// TIA Portal V17 export
// export: Created 2025-03-05T08:03:14.3285164Z, ExportSetting WithDefaults, DisplayName Totally Integrated Automation Portal, DisplayVersion V17 Update 8, DisplayName TIA Portal Openness, DisplayVersion V17 Update 8, DisplayName TIA Portal Version Control Interface, DisplayVersion V17, DisplayName SINAMICS Startdrive Advanced, DisplayVersion V17 SP2, DisplayName SINAMICS Startdrive G110M, G120, G120C, G120D, G120P, G115D, DisplayVersion V17 SP2, DisplayName SINAMICS Startdrive G130, G150, S120, S150, SINAMICS MV, S210, DisplayVersion V17 SP2, DisplayName STEP 7 Professional, DisplayVersion V17 Update 8, DisplayName SINUMERIK ONE STEP 7 Toolbox, DisplayVersion V17 Update 12, DisplayName SINUMERIK 840D sl STEP 7 Toolbox, DisplayVersion V17 Update 12, DisplayName STEP 7 Safety, DisplayVersion V17 Update 6, DisplayName WinCC Advanced, DisplayVersion V17 Update 8
FUNCTION_BLOCK "FB22102_POWDER_FLOW_SENSOR"   // FB22102, LAD
TITLE = FB22102 POWDER FLOW SENSOR
{ S7_Optimized_Access := 'FALSE' }
VERSION : 0.1
// stored: AutoNumber false, IsIECCheckEnabled false, SetENOAutomatically false, UDAEnableTagReadback false
   VAR_INPUT
      iANALOG_INPUT : UInt;
   END_VAR
   VAR_OUTPUT
      oPOWDER_FLOW_ON : Bool;
      oWARNING_LIMIT : Bool;
   END_VAR
   VAR DB_SPECIFIC
      OUTPUT : Struct
         VALUE : Real;
      END_STRUCT;
      INPUT_SETTINGS : Struct
         LOW_RANGE : Real;
         HIGH_RANGE : Real;
         LOW_LIM_TO_FLOW_ON : Real;
         UNIT_NUMBER : Int;
         HOPPER_NUMBER : Int;
      END_STRUCT;
      ALARM_SETTINGS : Struct
         WARN_LIMIT_LOW : Real;
         WARN_LIMIT_HIGH : Real;
         ERROR_CONFIGURATION : Bool;
      END_STRUCT;
      LOG : Struct
         SPARE : Bool;
      END_STRUCT;
   END_VAR
   VAR_TEMP
      DB_NUMBER : DInt;
      NORM_VALUE : Real;
   END_VAR
BEGIN

NETWORK
TITLE = READ INSTANCE DB NUMBER
      L     DINO;
      +     10#800000;
      T     #DB_NUMBER;

REGION Network 2: NORM AND SCALE ANALOG INPUT
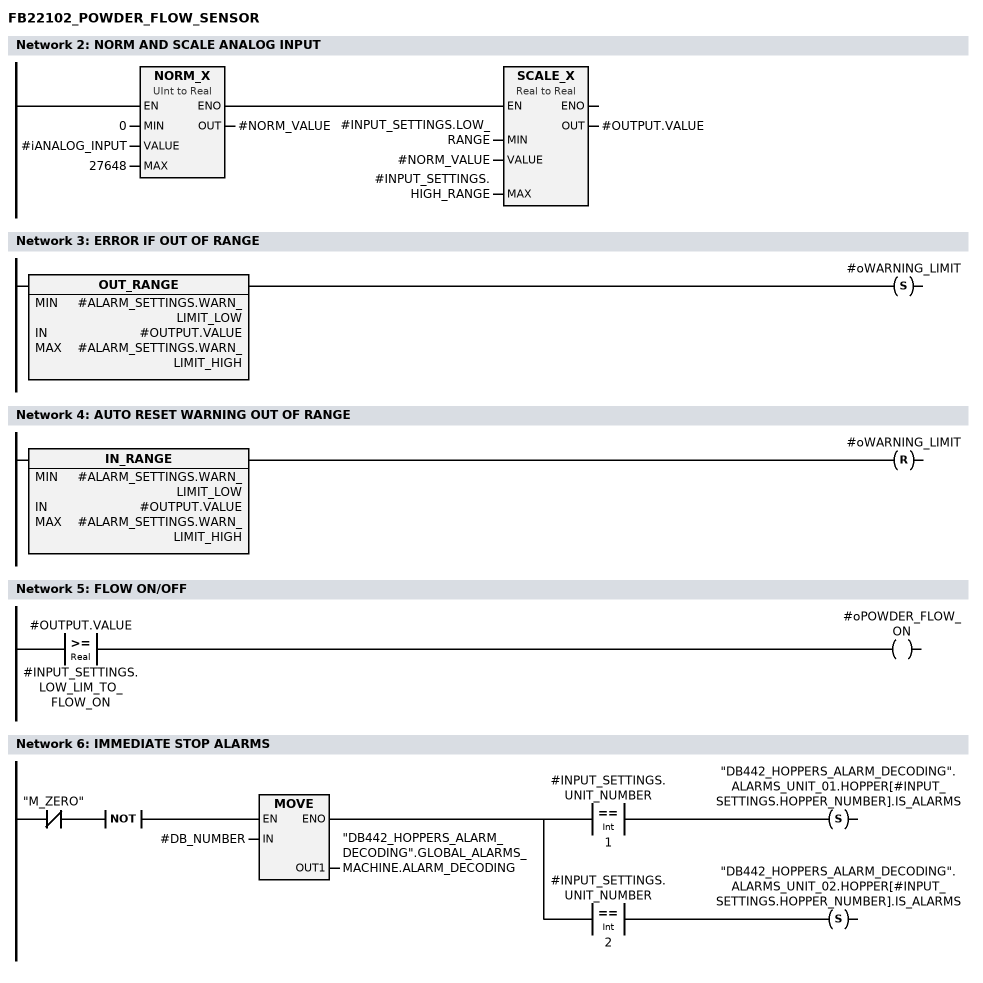
   RUNG wire#powerrail
      { S7_Templates := "[SrcType := UInt, DestType := Real]" } Normalize(min := 0, value := #iANALOG_INPUT, max := 27648, out => #NORM_VALUE)
      { S7_Templates := "[SrcType := Real, DestType := Real]" } Scale(min := #INPUT_SETTINGS.LOW_RANGE, value := #NORM_VALUE, max := #INPUT_SETTINGS.HIGH_RANGE, out => #OUTPUT.VALUE)
   END_RUNG
   // the same network as SCL:
   #NORM_VALUE := NORM_X(MIN := 0, VALUE := #iANALOG_INPUT, MAX := 27648);
   #OUTPUT.VALUE := SCALE_X(MIN := #INPUT_SETTINGS.LOW_RANGE, VALUE := #NORM_VALUE, MAX := #INPUT_SETTINGS.HIGH_RANGE);
END_REGION

REGION Network 3: ERROR IF OUT OF RANGE
   IF (#OUTPUT.VALUE < #ALARM_SETTINGS.WARN_LIMIT_LOW) OR (#OUTPUT.VALUE > #ALARM_SETTINGS.WARN_LIMIT_HIGH) THEN
       #oWARNING_LIMIT := TRUE;
   END_IF;
END_REGION

REGION Network 4: AUTO RESET WARNING OUT OF RANGE
   RUNG wire#powerrail
      { S7_Templates := "SrcType := Real" } InRange(min := #ALARM_SETTINGS.WARN_LIMIT_LOW, in := #OUTPUT.VALUE, max := #ALARM_SETTINGS.WARN_LIMIT_HIGH)
      R_Coil( #oWARNING_LIMIT )
   END_RUNG
   // the same network as SCL:
   IF (#ALARM_SETTINGS.WARN_LIMIT_LOW <= #OUTPUT.VALUE) AND (#OUTPUT.VALUE <= #ALARM_SETTINGS.WARN_LIMIT_HIGH) THEN
       #oWARNING_LIMIT := FALSE;
   END_IF;
END_REGION

REGION Network 5: FLOW ON/OFF
   RUNG wire#powerrail
      { S7_Templates := "SrcType := Real" } GE_Contact(in1 := #OUTPUT.VALUE, in2 := #INPUT_SETTINGS.LOW_LIM_TO_FLOW_ON)
      Coil( #oPOWDER_FLOW_ON )
   END_RUNG
   // the same network as SCL:
   #oPOWDER_FLOW_ON := #OUTPUT.VALUE >= #INPUT_SETTINGS.LOW_LIM_TO_FLOW_ON;
END_REGION

REGION Network 6: IMMEDIATE STOP ALARMS
   RUNG wire#powerrail
      I_Contact( "M_ZERO" )
      Not()
      { S7_GenerateENO := "TRUE" } Move(in := #DB_NUMBER, out1 => "DB442_HOPPERS_ALARM_DECODING".GLOBAL_ALARMS_MACHINE.ALARM_DECODING)
      wire#w1
      { S7_Templates := "SrcType := Int" } EQ_Contact(in1 := #INPUT_SETTINGS.UNIT_NUMBER, in2 := 1)
      S_Coil( "DB442_HOPPERS_ALARM_DECODING".ALARMS_UNIT_01.HOPPER[#INPUT_SETTINGS.HOPPER_NUMBER].IS_ALARMS )
   END_RUNG
   RUNG wire#w1
      { S7_Templates := "SrcType := Int" } EQ_Contact(in1 := #INPUT_SETTINGS.UNIT_NUMBER, in2 := 2)
      S_Coil( "DB442_HOPPERS_ALARM_DECODING".ALARMS_UNIT_02.HOPPER[#INPUT_SETTINGS.HOPPER_NUMBER].IS_ALARMS )
   END_RUNG
   // the same network as SCL:
   // ENO of a box is taken as its EN; it also drops when the box reports an error
   IF NOT (NOT "M_ZERO") THEN
       "DB442_HOPPERS_ALARM_DECODING".GLOBAL_ALARMS_MACHINE.ALARM_DECODING := #DB_NUMBER;
   END_IF;
   IF NOT (NOT "M_ZERO") AND (#INPUT_SETTINGS.UNIT_NUMBER = 1) THEN
       "DB442_HOPPERS_ALARM_DECODING".ALARMS_UNIT_01.HOPPER[#INPUT_SETTINGS.HOPPER_NUMBER].IS_ALARMS := TRUE;
   END_IF;
   IF NOT (NOT "M_ZERO") AND (#INPUT_SETTINGS.UNIT_NUMBER = 2) THEN
       "DB442_HOPPERS_ALARM_DECODING".ALARMS_UNIT_02.HOPPER[#INPUT_SETTINGS.HOPPER_NUMBER].IS_ALARMS := TRUE;
   END_IF;
END_REGION
END_FUNCTION_BLOCK
